(* CODESYS project util.library
   Company: TINEA
   Title: regulation
   Version: 0.0.0.0

Project tree, tasks and I/O mapping:
  libraries: Tc2_Standard, * (Beckhoff Automation GmbH)
  Data types/
    data type GEN_MODE
    data type POINT
  Global Variables/
    global variables Globale_Variablen
  POUs/
    analog monitors/
      function block HYSTERESIS [ST]
      function block LIMITALARM [ST]
    BCD CO_Nversions/
      function BCD_TO_INT [ST]
      function INT_TO_BCD [ST]
    bit_byte functions/
      function EXTRACT [ST]
      function PACK [ST]
      function PUTBIT [ST]
      function block UNPACK [ST]
    CO_Ntroller/
      function block PD [ST]
      function block PID [ST]
      function block PID_FIXCYCLE [ST]
    function manipulators/
      function block CHARCURVE [ST]
      function block RAMP_INT [ST]
      function block RAMP_REAL [ST]
    mathematical functions/
      function block DERIVATIVE [ST]
      function block INTEGRAL [ST]
      function block LIN_TRAFO [ST]
      function block STATISTICS_INT [ST]
      function block STATISTICS_REAL [ST]
      function block VARIANCE [ST]
    signals/
      function block BLINK [ST]
      function block FREQ_MEASURE [ST]
      function block GEN [ST]
    function Version_Util [ST]
  Visualizations/
*)

// Data types/GEN_MODE
TYPE GEN_MODE :
	(TRIANGLE:=0,TRIANGLE_POS:=1,SAWTOOTH_RISE:=2,SAWTOOTH_FALL:=3,RECTANGLE:=4,SINUS:=5,COSINUS:=6);
END_TYPE

// Data types/POINT
TYPE POINT :
STRUCT
	X,Y: DINT;
END_STRUCT
END_TYPE

// Global Variables/Globale_Variablen
{attribute 'Tc2GvlVarNames'}
VAR_GLOBAL
END_VAR

// POUs/BCD CO_Nversions/BCD_TO_INT
(* function reads BCD-Byte and returns its INT value; a wrong BCD value causes a return of -1 *)
FUNCTION BCD_TO_INT : INT
VAR_INPUT
	B:BYTE;		(* byte containing the BCD value *)
END_VAR

IF SHR(B,4)>9 OR B-SHL(SHR(B,4),4)>9 THEN
	BCD_TO_INT:=-1;
ELSE
	BCD_TO_INT:=B-SHR(B,4)*6;
END_IF;

END_FUNCTION

// POUs/signals/BLINK
FUNCTION_BLOCK BLINK
(* Function block to simulate a turn signal *)
VAR_INPUT
	ENABLE:BOOL;		(* TRUE:run Blink, FALSE: OUT keeps its value*)
	TIMELOW:TIME;		(* Time for OUT=FALSE *)
	TIMEHIGH:TIME;		(* Time for OUT=TRUE *)
END_VAR
VAR_OUTPUT
	OUT:BOOL;			(* output variable, starting with FALSE *)
END_VAR
VAR
	CLOCK:TP;
END_VAR

CLOCK();										(* call Timer *)
IF CLOCK.Q=FALSE AND ENABLE THEN	(* time passed or init *)
	CLOCK(IN:=FALSE);						(* reset Timer *)
	CLOCK(IN:=TRUE);						(* restart Timer *)
	IF OUT=FALSE THEN
		CLOCK.PT:=TIMEHIGH;
	ELSE
		CLOCK.PT:=TIMELOW;
	END_IF;
	OUT := NOT OUT;							(* invert *)
END_IF

END_FUNCTION_BLOCK

// POUs/function manipulators/CHARCURVE
(* function block to map an input signal on a characteristic curve *)
FUNCTION_BLOCK CHARCURVE
VAR_INPUT
	IN:INT;								(* input signal *)
	N:BYTE;							(* number of  points defining the characteristic curve : 2<=N<=11 *)
END_VAR
VAR_IN_OUT
	P:ARRAY[0..10] OF POINT;		(* ARRAY of N points to describe the characteristic curve *)
END_VAR
VAR_OUTPUT
	OUT:INT;							(* output variable *)
	ERR: BYTE;							(* error :
												0 : 	no error
												1 :	error in ARRAY: wrong sequence ( completely tested, only if IN is equal to largest X-value of P)
												2 :	IN outside of limits of P
												4 :	number of POINTS (N) invalid *)
END_VAR
VAR
	I:INT;
END_VAR

IF 1<N AND N<12 THEN							(* N zulässig ? *)
	ERR:=0;
	IF IN<P[0].X THEN							(* Prüfe, ob IN im zulässigen Bereich *)
		ERR:=2;
		OUT:=DINT_TO_INT(P[0].Y);
	ELSIF IN>P[N-1].X THEN						(* Prüfe, ob IN im zulässigen Bereich *)
		ERR:=2;
		OUT:=DINT_TO_INT(P[N-1].Y);
	ELSE
		FOR I:=1 TO N-1 DO
			IF P[I-1].X>=P[I].X THEN			(* Prüfe, ob Reihenfolge der Punkte richtig *)
				ERR:=1;
				EXIT;
			END_IF;
			IF IN<=P[I].X THEN					(* Verlasse Schleife, wenn IN im Intervall [I-1;I] *)
				EXIT;
			END_IF
		END_FOR;
		IF ERR=0 THEN
			OUT:=DINT_TO_INT(P[I].Y-(P[I].X-IN)*(P[I].Y-P[I-1].Y)/(P[I].X-P[I-1].X));	(* Berechne OUT *)
		ELSE
			OUT:=0;
		END_IF;
	END_IF
ELSE
	ERR:=4;
END_IF;

END_FUNCTION_BLOCK

// POUs/mathematical functions/DERIVATIVE
(* function block to approximate the derivative of a value *)
(* to calculate this, always four values are used in order to be as exact as possible *)
FUNCTION_BLOCK DERIVATIVE
VAR_INPUT
	IN:REAL;						(* input variable *)
	TM:DWORD;					(* time since last call in msec *)
	RESET:BOOL;					(* reset: set OUT to zero *)
END_VAR
VAR_OUTPUT
	OUT:REAL;					(* derivative *)
END_VAR
VAR
	X3,X2,X1:REAL;
	T2,T1:DWORD;
	INIT:BOOL:=TRUE;
END_VAR

IF INIT OR RESET THEN
	X1:=IN;
	X2:=IN;
	X3:=IN;
	OUT:=0;
	INIT:=FALSE;
ELSE
	IF TM>0 THEN
		OUT:=(3*(IN-X3)+X1-X2)/((3*T2+4*T1+3*TM))*1000;
		X3:=X2;
		X2:=X1;
		X1:=IN;
		T2:=T1;
		T1:=TM;
	END_IF;
END_IF;

END_FUNCTION_BLOCK

// POUs/bit_byte functions/EXTRACT
(* function returns Bit N of value X *)
FUNCTION EXTRACT : BOOL
VAR_INPUT
	X:DWORD;	(* value *)
	N:BYTE;		(* number of bit to be extracted *)
END_VAR
VAR
END_VAR

EXTRACT:=((SHR(X,N) AND 1)=1);

END_FUNCTION

// POUs/signals/FREQ_MEASURE
FUNCTION_BLOCK FREQ_MEASURE
(* FB to measure the frequency of a signal *)
VAR_INPUT
	IN:BOOL;						(* input signal *)
	PERIODS: INT (1..10) :=1;	(* out is the average frequency during PERIODS (number of periods) *)
	RESET: BOOL;				(* reset measurement *)
END_VAR
VAR_OUTPUT
	OUT:REAL;					(* frequency [Hz]*)
	VALID:BOOL;					(* FALSE: not yet PERIODS measurements done OR time distance between two rising edges > 3*OUT *)
END_VAR
VAR
	OLDIN: BOOL;
	INIT: BOOL;
	OLDT: TIME;
	DIFF: DWORD;
	ADIFF: ARRAY[0..9] OF DWORD;
	V: INT;
	B:INT;
	I: INT;
END_VAR

IF RESET THEN
	B:=0;
	V:=0;
	INIT:=FALSE;
	VALID:=FALSE;
	OUT:=0;
	RETURN;
END_IF

IF IN AND NOT OLDIN THEN	(*rising edge *)
	IF INIT THEN
		DIFF := TIME_TO_DWORD(TIME()-OLDT);
		IF Diff > 0 THEN
			ADIFF[B] := DIFF;
			B := (B+1) MOD PERIODS;
			V:= MIN(V+1, PERIODS);
			IF V=PERIODS THEN
				OUT := 0;
				FOR I:=0 TO PERIODS-1 DO
					OUT := OUT + ADIFF[I];
				END_FOR
				OUT := 1000.0 * PERIODS / OUT;
				VALID:=TRUE;
			ELSE
				VALID:=FALSE;
			END_IF
		END_IF
	END_IF
	INIT := TRUE;
	OLDT := TIME();
ELSIF INIT AND VALID AND TIME_TO_DWORD(TIME()-OLDT) > 3000*OUT THEN
	VALID:=FALSE;
	V:=0;
	B:=0;
END_IF

OLDIN:=IN;

END_FUNCTION_BLOCK

// POUs/signals/GEN
(* function block for generating some periodic functions *)
FUNCTION_BLOCK GEN
VAR_INPUT
	MODE:GEN_MODE;	(* define type :
								TRIANGLE				triangular	from - AMPL. to + AMPL.
								TRIANGLE_POS		triangular	from 0 to AMPL. 
								SAWTOOTH_RISE	sawtooth increasing from -AMPL. to +AMPL.
								SAWTOOTH_FALL	sawtooth decreasing from AMPL to -AMPL
								RECTANGLE			rectangular switching from  -AMPL. to +AMPL 
								SINUS					sinus
								COSINUS				cosinus *)
	BASE:BOOL;			(* FALSE: period referring to call; TRUE: period referring to time *)
	PERIOD:TIME:=t#1s;	(* period time, only relevant if BASE=TRUE *)
	CYCLES:INT:=1000;	(* number of calls per period, only relevant if BASE=FALSE *)
	AMPLITUDE:INT;		(* amplitude *)
	RESET:BOOL;			(* reset *)
END_VAR
VAR_OUTPUT
	OUT:INT;				(* generated function variable *)
END_VAR
VAR
	CET,PER:DINT;
	COUNTER:INT;
	CLOCK:TON;
	help: REAL;
END_VAR

IF RESET THEN
	COUNTER:=0;
	OUT:=0;
	CLOCK.PT := t#0s;
	CLOCK(IN:=FALSE);
ELSE
	IF BASE=FALSE THEN
		COUNTER:=(COUNTER+1)MOD CYCLES;
		CASE MODE OF
		0:	(* Dreiecksfunktion von -AMPL bis AMPL.*)
			OUT:=(CYCLES-2*ABS(CYCLES-2*COUNTER))*AMPLITUDE/CYCLES;
		1:	(* Dreiecksfunktion von 0 bis AMPL.*)
			OUT:=(CYCLES-ABS(CYCLES-2*COUNTER))*AMPLITUDE/CYCLES;
		2:	(* Sägezahn steigend *)
			OUT:=(2*COUNTER-CYCLES)*AMPLITUDE/CYCLES;
		3:	(* Sägezahn fallend *)
			OUT:=(CYCLES-2*COUNTER)*AMPLITUDE/CYCLES;
		4:	(* Rechteck AMPL./-AMPL. *)
			IF 2*COUNTER>CYCLES THEN
				OUT:=-AMPLITUDE;
			ELSE
				OUT:=AMPLITUDE;
			END_IF
		5:	(* Sinusfunktion *)
			help := 6.283167*COUNTER/CYCLES;
			OUT:=LREAL_TO_INT(SIN(help)*AMPLITUDE);
		6:	(* Cosinusfunktion *)
			help := 6.283167*COUNTER/CYCLES;
			OUT:=LREAL_TO_INT(COS(help)*AMPLITUDE);
		END_CASE;
	ELSE										(* Periodizität bzgl. Zeit *)
				CLOCK();									(* Timer abfragen *)
		IF CLOCK.PT<>PERIOD+PERIOD THEN			(* Initialisierung *)
			CLOCK.PT:=PERIOD+PERIOD;			(* Setze Timer auf zwei PERIODn *)
			CLOCK(IN:=TRUE);
		ELSE
			CET:=TIME_TO_DINT(CLOCK.ET);
			PER:=TIME_TO_DINT(PERIOD);
			IF CET>=PER THEN					(* Neuinitialisierung des Timers *)
				CLOCK(IN:=FALSE);
				CLOCK(IN:=TRUE);
				CET:=CET MOD PER;
			END_IF
			CASE MODE OF
			0:	(* Dreiecksfunktion -AMPL bis AMPL.*)
				OUT:=DINT_TO_INT((2*ABS(PER-2*CET)*AMPLITUDE+PER/2)/PER-AMPLITUDE);
			1:	(* Dreiecksfunktion 0 bis AMPL.*)
				OUT:=DINT_TO_INT(((PER-ABS(PER-2*CET))*AMPLITUDE+PER/2)/PER);
			2:	(* Sägezahn steigend *)
				OUT:=DINT_TO_INT((CET-PER)*2*AMPLITUDE/PER+AMPLITUDE);
			3:	(* Sägezahn fallend *)
				OUT:=DINT_TO_INT((PER-CET)*2*AMPLITUDE/PER+AMPLITUDE);
			4:	(* Rechteck AMPL./-AMPL. *)
				IF CET*2<PER THEN
					OUT:=-AMPLITUDE;
				ELSE
					OUT:=AMPLITUDE;
				END_IF
			5:	(* Sinusfunktion *)
				help := 6.283167*CET;
				help:=SIN(help/PER)*AMPLITUDE;
				OUT:=REAL_TO_INT(help+0.5);
			6:	(* Cosinusfunktion *)
				help := 6.283167*CET;
				help:=COS(help/PER)*AMPLITUDE;
				OUT:=LREAL_TO_INT(help+0.5);
			END_CASE;
		END_IF
	END_IF;
END_IF;

END_FUNCTION_BLOCK

// POUs/analog monitors/HYSTERESIS
(* function block, which sets OUT to TRUE, if input IN is less than LOW, and which sets OUT to FALSE, if input IN is bigger than HIGH *)
FUNCTION_BLOCK HYSTERESIS
VAR_INPUT
	IN:INT;			(* input value *)
	HIGH:INT;		(* upper threshold value *)
	LOW:INT;		(* lower threshold value *)
END_VAR
VAR_OUTPUT
	OUT:BOOL;	(* hysteresis value *)
END_VAR
VAR
END_VAR

IF  IN<LOW THEN
	OUT:=TRUE;
END_IF;
IF IN>HIGH THEN
	OUT:=FALSE;
END_IF;

END_FUNCTION_BLOCK

// POUs/BCD CO_Nversions/INT_TO_BCD
(* function reads INT and returns its BCD value; a wrong INT value (<0 or >99) causes a return of 255 *)
FUNCTION INT_TO_BCD : BYTE
VAR_INPUT
	I:INT;		(* INT value to be converted to BCD*)
END_VAR
VAR
END_VAR

IF I>99 OR I<0 THEN
	INT_TO_BCD:=255;
ELSE
	INT_TO_BCD:=INT_TO_BYTE((I/10)*6+I);
END_IF;

END_FUNCTION

// POUs/mathematical functions/INTEGRAL
(* function block to approximate the integral of IN over the time *)
FUNCTION_BLOCK INTEGRAL
VAR_INPUT
	IN:REAL;						(* input variable *)
	TM:DWORD;					(* time since last call in msec *)
	RESET:BOOL;					(* reset: OUT is set to zero and OVERFLOW to false *)
END_VAR
VAR_OUTPUT
	OUT:REAL;					(* value of the integral *)
	OVERFLOW:BOOL:=FALSE;	(* overflow *)
END_VAR
VAR
END_VAR

IF RESET THEN
	OUT:=0;
	OVERFLOW:=FALSE;
ELSIF NOT OVERFLOW  THEN
	IF 1E38 - IN*TM < OUT OR -1E38 - IN*TM > OUT THEN
		OVERFLOW:=TRUE;
	ELSE
		OUT:=OUT+IN*TM/1000;
	END_IF;
END_IF;

END_FUNCTION_BLOCK

// POUs/analog monitors/LIMITALARM
(* function block monitoring, whether the input value IN lies between LOW and HIGH *)
FUNCTION_BLOCK LIMITALARM
VAR_INPUT
	IN:INT;					(* INPUT value *)
	HIGH:INT;				(* upper threshold value *)
	LOW:INT;				(* lower threshold value *)
END_VAR
VAR_OUTPUT
	O:BOOL;				(* TRUE, if IN > HIGH, else FALSE *)
	U:BOOL;				(* TRUE, if IN < LOW, else FALSE *)
	IL:BOOL;				(* neither O nor U *)
END_VAR
VAR
END_VAR

O:=(IN>HIGH);
U:=(IN<LOW);
IL:=NOT (O OR U);

END_FUNCTION_BLOCK

// POUs/mathematical functions/LIN_TRAFO
(* linear transformation *)
FUNCTION_BLOCK LIN_TRAFO
VAR_INPUT
	IN: REAL;				(* input value*)
	IN_MIN:REAL;			(* minimum input value *)
	IN_MAX:REAL;			(* maximum input value *)
	OUT_MIN:REAL;		(* corresponding minimum output value *)
	OUT_MAX:REAL;		(* corresponding maximum output value *)
END_VAR
VAR_OUTPUT
	OUT: REAL;			(* output value *)
	ERROR: BOOL;		(* error: IN_MIN = IN_MAX or IN out of interval *)
END_VAR

VAR
	Diff: REAL;
END_VAR

Diff := IN_MAX-IN_MIN;
ERROR := (Diff=0) OR (IN<IN_MIN) OR (IN>IN_MAX);

IF NOT ERROR THEN
	OUT := (IN-IN_MIN)/Diff * (OUT_MAX-OUT_MIN) + OUT_MIN;
END_IF

END_FUNCTION_BLOCK

// POUs/bit_byte functions/PACK
(* pack eight bits into 1 byte *)
FUNCTION PACK : BYTE
VAR_INPUT
	B0:BOOL;		(* value of bit 0 *)
	B1:BOOL;		(* value of bit 1 *)
	B2:BOOL;		(* value of bit 2 *)
	B3:BOOL;		(* value of bit 3 *)
	B4:BOOL;		(* value of bit 4 *)
	B5:BOOL;		(* value of bit 5 *)
	B6:BOOL;		(* value of bit 6 *)
	B7:BOOL;		(* value of bit 7 *)
END_VAR

PACK:=BOOL_TO_BYTE(B7);
PACK:=PACK*2+BOOL_TO_BYTE(B6);
PACK:=PACK*2+BOOL_TO_BYTE(B5);
PACK:=PACK*2+BOOL_TO_BYTE(B4);
PACK:=PACK*2+BOOL_TO_BYTE(B3);
PACK:=PACK*2+BOOL_TO_BYTE(B2);
PACK:=PACK*2+BOOL_TO_BYTE(B1);
PACK:=PACK*2+BOOL_TO_BYTE(B0);

END_FUNCTION

// POUs/CO_Ntroller/PD
(* PD controller *)
FUNCTION_BLOCK PD
VAR_INPUT
	ACTUAL :REAL;		(* actual value, process variable *)
	SET_POINT:REAL;	(* desired value, set point *)
	KP:REAL;				(* proportionality const. (P)*)
	TV:REAL;				(* rate time, derivative time (D) in sec *)
	Y_MANUAL:REAL;		(* Y is set to this value as long as MANUAL=TRUE *)
	Y_OFFSET:REAL;		(* offset for manipulated variable *)
	Y_MIN:REAL;			(* minimum value for manipulated variable *)
	Y_MAX:REAL;			(* maximum value for manipulated variable *)
	MANUAL:BOOL;		(* 	TRUE: manual: Y is not influenced by controller,
								FALSE: controller determines Y *)
	RESET:BOOL;			(* reset: set Y output to Y_OFFSET *)
END_VAR
VAR_OUTPUT
	Y:REAL;				(* manipulated variable, set value*)
	LIMITS_ACTIVE:BOOL:=FALSE;	(* true set value would exceed limits Y_MIN, Y_MAX *)
END_VAR
VAR
	CLOCK:TON;
	D: DERIVATIVE;
	TMDIFF: DWORD;
	ERROR: REAL;
	INIT: BOOL:=TRUE;
	Y_ADDOFFSET: REAL;
	KPcopy:REAL;
	TVcopy:REAL;
END_VAR

IF KP<> 0 THEN
	ERROR := SET_POINT-ACTUAL;								(* Regeldifferenz *)

	IF RESET OR MANUAL OR INIT OR (KP<>KPcopy OR TV<>TVcopy) THEN							(* Reset oder Handbetrieb *)
		D(RESET:=TRUE);
		LIMITS_ACTIVE:=FALSE;
		IF RESET OR INIT THEN
			Y := Y_OFFSET;
			INIT:=FALSE;
			Y_ADDOFFSET :=  0;
		ELSIF MANUAL THEN
			Y := Y_MANUAL;
			Y_ADDOFFSET := Y_MANUAL-(Y_OFFSET+KP*(ERROR+D.OUT*TV));
		ELSE
			Y_ADDOFFSET := Y - Y_OFFSET - KP*ERROR;
		END_IF
		TMDIFF:=0;
		CLOCK(IN:=FALSE);									(* Timer neu starten *)
		CLOCK(PT:=t#1h, IN:=TRUE);

		TVcopy := TV;
		KPcopy := KP;
	ELSE
				CLOCK();												(* Timer abfragen *)
		TMDIFF:=TIME_TO_DWORD(CLOCK.ET);					(* Zeitdifferenz seit letztem Aufruf *)
	END_IF;

	IF TMDIFF>0 THEN
		CLOCK(IN:=FALSE);									(* Timer neu starten *)
		CLOCK(PT:=t#1h, IN:=TRUE);

		D(IN:=ERROR, TM:=TMDIFF, RESET:=FALSE);				(* Differential abschätzen *)

		Y:=Y_OFFSET+KP*(ERROR+D.OUT*TV) + Y_ADDOFFSET;

		LIMITS_ACTIVE:=FALSE;
		IF Y_MAX>Y_MIN AND Y>Y_MAX  THEN					(* Stellwert-Obergrenze überschritten *)
			Y:=Y_MAX;
			LIMITS_ACTIVE:=TRUE;
		END_IF;

		IF Y_MAX>Y_MIN AND Y<Y_MIN THEN						(* Stellwert-Untergrenze unterschritten *)
			Y:=Y_MIN;
			LIMITS_ACTIVE:=TRUE;
		END_IF;
	ELSE
		CLOCK(PT:=t#1h,IN:=TRUE);
	END_IF;

END_IF;

END_FUNCTION_BLOCK

// POUs/CO_Ntroller/PID
(* PD controller *)
FUNCTION_BLOCK PID
VAR_INPUT
	ACTUAL :REAL;		(* actual value, process variable *)
	SET_POINT:REAL;	(* desired value, set point *)
	KP:REAL;				(* proportionality const. (P)*)
	TN:REAL;				(* reset time (I) in sec *)
	TV:REAL;				(* rate time, derivative time (D) in sec*)
	Y_MANUAL:REAL;		(* Y is set to this value as long as MANUAL=TRUE *)
	Y_OFFSET:REAL;		(* offset for manipulated variable *)
	Y_MIN:REAL;			(* minimum value for manipulated variable *)
	Y_MAX:REAL;			(* maximum value for manipulated variable *)
	MANUAL:BOOL;		(* 	TRUE: manual: Y is not influenced by controller,
								FALSE: controller determines Y *)
	RESET:BOOL;			(* reset: set Y output to Y_OFFSET and reset integral part *)
END_VAR
VAR_OUTPUT
	Y:REAL;				(* manipulated variable, set value*)
	LIMITS_ACTIVE:BOOL:=FALSE;	(* true set value would exceed limits Y_MIN, Y_MAX *)
	OVERFLOW:BOOL:=FALSE;		(* overflow in integral part *)
END_VAR
VAR
	CLOCK:TON;
	I: INTEGRAL;
	D: DERIVATIVE;
	TMDIFF: DWORD;
	ERROR: REAL;
	INIT: BOOL:=TRUE;
	Y_ADDOFFSET: REAL;
	KPcopy:REAL;
	TNcopy:REAL;
	TVcopy:REAL;
END_VAR

IF TN>0 AND KP<> 0 AND (NOT OVERFLOW OR RESET OR MANUAL) THEN
	ERROR := SET_POINT-ACTUAL;								(* Regeldifferenz *)

	IF RESET OR MANUAL OR INIT OR (KP<>KPcopy OR TN<>TNcopy OR TV<>TVcopy) THEN							(* Reset oder Handbetrieb *)
		I(RESET:=TRUE);
		D(RESET:=TRUE);
		OVERFLOW:=FALSE;
		LIMITS_ACTIVE:=FALSE;
		IF RESET OR INIT THEN
			Y := Y_OFFSET;
			INIT:=FALSE;
			Y_ADDOFFSET := 0;
		ELSIF MANUAL THEN
			Y := Y_MANUAL;
			Y_ADDOFFSET := Y_MANUAL-(Y_OFFSET+KP*(ERROR+I.OUT/TN+D.OUT*TV));
		ELSE
			Y_ADDOFFSET := Y - Y_OFFSET - KP*ERROR;
		END_IF
		TMDIFF:=0;
		CLOCK(IN:=FALSE);									(* Timer neu starten *)
		CLOCK(PT:=t#1h, IN:=TRUE);

		TNcopy := TN;
		TVcopy := TV;
		KPcopy := KP;
	ELSE
				CLOCK();												(* Timer abfragen *)
		TMDIFF:=TIME_TO_DWORD(CLOCK.ET);					(* Zeitdifferenz seit letztem Aufruf *)
	END_IF;

	IF TMDIFF>0 THEN
		CLOCK(IN:=FALSE);									(* Timer neu starten *)
		CLOCK(PT:=t#1h, IN:=TRUE);

		D(IN:=ERROR, TM:=TMDIFF, RESET:=FALSE);				(* Differential abschätzen *)
		I(IN:=ERROR, TM:=TMDIFF, RESET:=FALSE);				(* Integral abschätzen *)

		OVERFLOW := I.OVERFLOW;
		IF NOT OVERFLOW THEN
			Y:=Y_OFFSET+KP*(ERROR+I.OUT/TN+D.OUT*TV) + Y_ADDOFFSET;
			IF Y>1E30 OR Y<-1E30 THEN						(* Overflow steht bevor, darf aber eigentlich nicht passieren *)
				OVERFLOW:=TRUE;
			END_IF;

			LIMITS_ACTIVE:=FALSE;
			IF Y_MAX>Y_MIN AND Y>Y_MAX  THEN				(* Stellwert-Obergrenze überschritten *)
				LIMITS_ACTIVE:=TRUE;
				IF KP<>0 THEN
					I(IN:=(Y_MAX-Y)*TN/KP,TM:=1000,RESET:=FALSE);		(* Integral korrigieren *)
				END_IF
				Y:=Y_MAX;
			END_IF;
			IF Y_MAX>Y_MIN AND Y<Y_MIN THEN					(* Stellwert-Untergrenze unterschritten *)
				LIMITS_ACTIVE:=TRUE;
				IF KP<>0 THEN
					I(IN:=(Y_MIN-Y)*TN/KP,TM:=1000,RESET:=FALSE);		(* Integral korrigieren *)
				END_IF
				Y:=Y_MIN;
			END_IF;
		END_IF;
	ELSE
		CLOCK(PT:=t#1h,IN:=TRUE);
	END_IF;

END_IF;

END_FUNCTION_BLOCK

// POUs/CO_Ntroller/PID_FIXCYCLE
(* PD controller *)
FUNCTION_BLOCK PID_FIXCYCLE
VAR_INPUT
	ACTUAL :REAL;		(* actual value, process variable *)
	SET_POINT:REAL;	(* desired value, set point *)
	KP:REAL;				(* proportionality const. (P)*)
	TN:REAL;				(* reset time (I) in sec *)
	TV:REAL;				(* rate time, derivative time (D) in sec*)
	Y_MANUAL:REAL;		(* Y is set to this value as long as MANUAL=TRUE *)
	Y_OFFSET:REAL;		(* offset for manipulated variable *)
	Y_MIN:REAL;			(* minimum value for manipulated variable *)
	Y_MAX:REAL;			(* maximum value for manipulated variable *)
	MANUAL:BOOL;		(* 	TRUE: manual: Y is not influenced by controller,
								FALSE: controller determines Y *)
	RESET:BOOL;			(* reset: set Y output to Y_OFFSET and reset integral part *)
	CYCLE:REAL;			(* time in s between two calls *)
END_VAR
VAR_OUTPUT
	Y:REAL;				(* manipulated variable, set value*)
	LIMITS_ACTIVE:BOOL:=FALSE;	(* true set value would exceed limits Y_MIN, Y_MAX *)
	OVERFLOW:BOOL:=FALSE;		(* overflow in integral part *)
END_VAR
VAR
	I: INTEGRAL;
	D: DERIVATIVE;
	TMDIFF: DWORD;
	ERROR: REAL;
	INIT: BOOL:=TRUE;
	Y_ADDOFFSET: REAL;
	KPcopy:REAL;
	TNcopy:REAL;
	TVcopy:REAL;
END_VAR

IF TN>0 AND KP<> 0 AND (NOT OVERFLOW OR RESET OR MANUAL) THEN
	ERROR := SET_POINT-ACTUAL;								(* Regeldifferenz *)

	IF RESET OR MANUAL OR INIT OR (KP<>KPcopy OR TN<>TNcopy OR TV<>TVcopy) THEN							(* Reset oder Handbetrieb *)
		I(RESET:=TRUE);
		D(RESET:=TRUE);
		OVERFLOW:=FALSE;
		LIMITS_ACTIVE:=FALSE;
		IF RESET OR INIT THEN
			Y := Y_OFFSET;
			INIT:=FALSE;
			Y_ADDOFFSET := 0;
		ELSIF MANUAL THEN
			Y := Y_MANUAL;
			Y_ADDOFFSET := Y_MANUAL-(Y_OFFSET+KP*(ERROR+I.OUT/TN+D.OUT*TV));
		ELSE
			Y_ADDOFFSET := Y - Y_OFFSET - KP*ERROR;
		END_IF
		TMDIFF:=0;

		TNcopy := TN;
		TVcopy := TV;
		KPcopy := KP;
	ELSE
		tmDiff:=REAL_TO_DWORD(CYCLE*1000);
	END_IF;

	IF TMDIFF>0 THEN

		D(IN:=ERROR, TM:=TMDIFF, RESET:=FALSE);				(* Differential abschätzen *)
		I(IN:=ERROR, TM:=TMDIFF, RESET:=FALSE);				(* Integral abschätzen *)

		OVERFLOW := I.OVERFLOW;
		IF NOT OVERFLOW THEN
			Y:=Y_OFFSET+KP*(ERROR+I.OUT/TN+D.OUT*TV) + Y_ADDOFFSET;
			IF Y>1E30 OR Y<-1E30 THEN						(* Overflow steht bevor, darf aber eigentlich nicht passieren *)
				OVERFLOW:=TRUE;
			END_IF;

			LIMITS_ACTIVE:=FALSE;
			IF Y_MAX>Y_MIN AND Y>Y_MAX  THEN				(* Stellwert-Obergrenze überschritten *)
				LIMITS_ACTIVE:=TRUE;
				IF KP<>0 THEN
					I(IN:=(Y_MAX-Y)*TN/KP,TM:=1000,RESET:=FALSE);		(* Integral korrigieren *)
				END_IF
				Y:=Y_MAX;
			END_IF;

			IF Y_MAX>Y_MIN AND Y<Y_MIN THEN					(* Stellwert-Untergrenze unterschritten *)
				LIMITS_ACTIVE:=TRUE;
				IF KP<>0 THEN
					I(IN:=(Y_MIN-Y)*TN/KP,TM:=1000,RESET:=FALSE);		(* Integral korrigieren *)
				END_IF
				Y:=Y_MIN;
			END_IF;
		END_IF;
	END_IF;

END_IF;

END_FUNCTION_BLOCK

// POUs/bit_byte functions/PUTBIT
(* function sets bit N of X to B and returns new value *)
FUNCTION PUTBIT : DWORD
VAR_INPUT
	X:DWORD;	(* value to be manipulated *)
	N:BYTE;		(* position of bit to be changed *)
	B:BOOL;		(* value of specified bit *)
END_VAR

IF B=TRUE THEN
	PUTBIT:=(X OR SHL(DWORD#1,N));
ELSE
	PUTBIT:=(X AND ROL(DWORD#4294967294,N));
END_IF;

END_FUNCTION

// POUs/function manipulators/RAMP_INT
(* function block to limit the slope of a value to a certain value *)
FUNCTION_BLOCK RAMP_INT
VAR_INPUT
	IN: INT;							(* input variable *)
	ASCEND: INT;						(* maximum positive slope *)
	DESCEND: INT;					(* maximum negative slope (non-negative!!) *)
	TIMEBASE: TIME;					(* reference for ASCEND/DESCEND :
											t#0s : ASCEND/DESCEND defined per call
											else : ASCEND/DESCEND defined per specified time*)
	RESET:BOOL;						(* reset *)
END_VAR
VAR_OUTPUT
	OUT: INT;							(* value of function with limited slope *)
END_VAR
VAR
	DIFF: DINT;
	OLD_IN: INT;
	TB,CET:DWORD;
	CH:INT;
	CLOCK: TON;
END_VAR

IF RESET=TRUE OR CLOCK.PT<>TIMEBASE THEN			(* Reset *)
	OLD_IN:=IN;
	CLOCK(PT:=TIMEBASE,IN:=FALSE);
END_IF

DIFF:=INT_TO_DINT(IN)-OLD_IN;									(* Änderung zum letzten WERT *)

IF TIMEBASE=t#0s THEN								(* Bezugswert : Aufruf *)
	IF DIFF>ASCEND THEN
		OUT:=OLD_IN+ASCEND;
	ELSIF DIFF<-DESCEND THEN
		OUT:=OLD_IN-DESCEND;
	ELSE
		OUT:=IN;
	END_IF;
ELSE												(* Bezugswert : TIMEBASE *)
	TB:=TIME_TO_DWORD(TIMEBASE);					(* TIMEBASE als DWORD *)
		CLOCK();
	CET:=TIME_TO_DWORD(CLOCK.ET);					(* verstrichene Zeit *)
	IF CET>0 THEN									(* wenn Zeit verstrichen *)
		IF (DWORD_TO_DINT(TB)*DIFF+CET/2)/DWORD_TO_DINT(CET)>ASCEND THEN			(* zu starker Anstieg *)
			CH:=DWORD_TO_INT((CET*ASCEND)/TB);
			IF CH<>0 THEN
					OUT:=OLD_IN+CH;
			END_IF;
		ELSIF DIFF*TB/DWORD_TO_DINT(CET)<-DESCEND THEN	(* zu starker Abfall *)
			CH:=DWORD_TO_INT((CET*DESCEND)/TB);
			IF CH<>0 THEN
					OUT:=OLD_IN-CH;
			END_IF;
		ELSE
			CH:=1;									(* Änderung in erlaubten Grenzen *)
			OUT:=IN;
		END_IF;
		IF CH<>0 THEN
			CLOCK(IN:=FALSE);						(* Timer neu starten *)
			CLOCK(IN:=TRUE);
		END_IF;
	ELSE											(* keine Zeit verstrichen *)
		CLOCK.PT:=TIMEBASE;							(* => ggf. Initialisierung *)
		CLOCK(IN:=TRUE);							(* => ggf. Timer neu starten *)
	END_IF;
END_IF;

OLD_IN:=OUT;

END_FUNCTION_BLOCK

// POUs/function manipulators/RAMP_REAL
(* function block to limit the slope of a value to a certain value *)
FUNCTION_BLOCK RAMP_REAL
VAR_INPUT
	IN: REAL;							(* input variable *)
	ASCEND: REAL;					(* maximum positive slope *)
	DESCEND: REAL;				(* maximum negative slope (non-negative!!) *)
	TIMEBASE: TIME;					(* reference for ASCEND/DESCEND :
											t#0s : ASCEND/DESCEND defined per call
											else : ASCEND/DESCEND defined per specified time*)
	RESET:BOOL;						(* reset *)
END_VAR
VAR_OUTPUT
	OUT: REAL;						(* value of function with limited slope *)
END_VAR
VAR
	DIFF: REAL;
	OLD_IN: REAL;
	TB,CET:DWORD;
	CLOCK: TON;
	probe:REAL;
END_VAR

IF RESET=TRUE OR CLOCK.PT<>TIMEBASE THEN			(* Reset *)
	OLD_IN:=IN;
	CLOCK(PT:=TIMEBASE,IN:=FALSE);
END_IF

DIFF:=IN-OLD_IN;									(* Änderung zum letzten WERT *)

IF TIMEBASE=t#0s THEN								(* Bezugswert : Aufruf *)
	IF DIFF>ASCEND THEN
		OUT:=OLD_IN+ASCEND;
	ELSIF DIFF<-DESCEND THEN
		OUT:=OLD_IN-DESCEND;
	ELSE
		OUT:=IN;
	END_IF;
ELSE												(* Bezugswert : TIMEBASE *)
	TB:=TIME_TO_DWORD(TIMEBASE);					(* TIMEBASE als DWORD *)
		CLOCK();
	CET:=TIME_TO_DWORD(CLOCK.ET);					(* verstrichene Zeit *)
	IF CET>0 THEN									(* wenn Zeit verstrichen *)
		CLOCK(IN:=FALSE);							(* Timer neu starten *)
		CLOCK(IN:=TRUE);
		probe:=DIFF*TB/CET;
		IF probe>ASCEND THEN						(* zu starker Anstieg *)
			OUT:=OLD_IN+ASCEND*CET/DWORD_TO_REAL(TB);
		ELSIF probe<-DESCEND THEN					(* zu starker Abfall *)
			OUT:=OLD_IN-DESCEND*CET/DWORD_TO_REAL(TB);
		ELSE										(* Änderung in erlaubten Grenzen *)
			OUT:=IN;
		END_IF;
	ELSE											(* keine Zeit verstrichen *)
		CLOCK.PT:=TIMEBASE;							(* => ggf. Initialisierung *)
		CLOCK(IN:=TRUE);							(* => ggf. Timer neu starten *)
	END_IF;
END_IF;

OLD_IN:=OUT;

END_FUNCTION_BLOCK

// POUs/mathematical functions/STATISTICS_INT
(* function block for statistics: calculating minimum, maximum and average of an input value *)
FUNCTION_BLOCK STATISTICS_INT
VAR_INPUT
	IN: INT;				(* input value*)
	RESET: BOOL;		(* reset: average set to 0, min and max to minimum and maximum possible INTs*)
END_VAR
VAR_OUTPUT
	MN: INT:=32767;		(* minimum value*)
	MX: INT:=-32768;		(* maximum value*)
	AVG: INT;				(* average value*)
END_VAR
VAR
	SUM:DINT;
	COUNTER:DINT;
END_VAR

IF RESET THEN
	AVG:=IN;
	COUNTER:=0;
	SUM:=0;
	MN:=IN;
	MX:=IN;
ELSE
	IF IN<MN THEN
		MN:=IN;
	END_IF
	IF IN>MX THEN
		MX:=IN;
	END_IF
	IF ABS(SUM)>2000000000 OR ABS(COUNTER)>2000000000 THEN		(* falls Überlauf droht *)
		SUM:=SUM/2;
		COUNTER:=COUNTER/2;
	END_IF;

	COUNTER:=COUNTER+1;
	SUM:=SUM+IN;
	AVG:=DINT_TO_INT((SUM+COUNTER/2)/COUNTER);  				(* gerundeter Durchschnitt *)
END_IF;

END_FUNCTION_BLOCK

// POUs/mathematical functions/STATISTICS_REAL
(* function block for statistics: calculating minimum, maximum and average of an input value *)
FUNCTION_BLOCK STATISTICS_REAL
VAR_INPUT
	IN: REAL;					(* input value*)
	RESET: BOOL;			(* reset: average set to 0, min and max to minimum and maximum possible REALs*)
END_VAR
VAR_OUTPUT
	MN: REAL:=3E+38;		(* minimum value*)
	MX: REAL:=1E-37;			(* maximum value*)
	AVG: REAL;				(* average value*)
END_VAR
VAR
	COUNTER: DINT;
	SUM:REAL;
END_VAR

IF RESET THEN
	AVG:=0;
	COUNTER:=0;
	SUM:=0;
	MN:=3.402823466e+38;
	MX:=1.175494351e-38;
ELSE
	IF IN<MN THEN
		MN:=IN;
	END_IF
	IF IN>MX THEN
		MX:=IN;
	END_IF

	IF ABS(COUNTER)>2000000000 THEN						(* falls Überlauf droht *)
		COUNTER:=COUNTER/2;
	END_IF;

	COUNTER:=COUNTER+1;
	AVG:=AVG/COUNTER*(COUNTER-1)+IN/COUNTER;
END_IF;

END_FUNCTION_BLOCK

// POUs/bit_byte functions/UNPACK
(* function block unpacks byte into 8 bits *)
FUNCTION_BLOCK UNPACK
VAR_INPUT
	B:BYTE;	(* byte to be unpacked *)
END_VAR
VAR_OUTPUT
	B0:BOOL;		(* value of bit 0 *)
	B1:BOOL;		(* value of bit 1 *)
	B2:BOOL;		(* value of bit 2 *)
	B3:BOOL;		(* value of bit 3 *)
	B4:BOOL;		(* value of bit 4 *)
	B5:BOOL;		(* value of bit 5 *)
	B6:BOOL;		(* value of bit 6 *)
	B7:BOOL;		(* value of bit 7 *)
END_VAR
VAR
END_VAR

B7:=BYTE_TO_BOOL(B AND 128);
B6:=BYTE_TO_BOOL(B AND 64);
B5:=BYTE_TO_BOOL(B AND 32);
B4:=BYTE_TO_BOOL(B AND 16);
B3:=BYTE_TO_BOOL(B AND 8);
B2:=BYTE_TO_BOOL(B AND 4);
B1:=BYTE_TO_BOOL(B AND 2);
B0:=BYTE_TO_BOOL(B AND 1);

END_FUNCTION_BLOCK

// POUs/mathematical functions/VARIANCE
(* function block to calculate the mathematical variance of a variable*)
FUNCTION_BLOCK VARIANCE
VAR_INPUT
	IN:REAL;		(* input variable *)
	RESET:BOOL;	(* reset *)
END_VAR
VAR_OUTPUT
	OUT:REAL;	(* variance *)
END_VAR
VAR
	Z:INT;
	A,B:REAL;
END_VAR

IF RESET THEN
	Z:=0;
	A:=0;
	B:=0;
	OUT:=0;
ELSE
	Z:=Z+1;
	A:=A+IN*IN;
	B:=B+IN;
	OUT:=(A-B*B/Z)/Z;
END_IF;

END_FUNCTION_BLOCK

// POUs/Version_Util
FUNCTION Version_Util : WORD
VAR_INPUT
	B:BOOL;
END_VAR
VAR
END_VAR
(******************************************************************************************)
(* Version,  Datum	Kommentar											*)
(* 1.00	28.02.2001	generated								 			*)
(* 1.01	29.06.2001	bugfix in GEN (HP)									*)
(* 1.02	03.01.2002	INTEGRAL was calculated for sec instead of msec 	*)
(* 1.03 	12.11.2002	comments added *)
(* 1.04 	23.01.2003	GEN:initial values for PERIOD and CYCLES to avoid div by zero *)
(* 1.05	13.06.2003	DERIVATIVE was calculated for sec instead of msec *)
(*	ATTENTION		TV/TN inputs of PD and PID refer to sec instead of msec *)
(* 1.06	25.06.2003	PD/PID: input Y_MANUAL added *)
(* 1.07	13.10.2003	PID_FIXCYCLE added *)
(* 1.08	09.01.2004	CHARCURVE: overflow fixed *)
(* 1.09	30.01.2004	GEN: if time based, reset induced freeze *)
(* 1.10	12.02.2004	all libs except standard.lib removed *)
(* 1.11	11.03.2005	PID: avoid jumps in Y (when limits change) by correcting integral part ; LIN_TRAFO added*)
(* 1.12	14.03.2005	FREQ_MEASURE added *)
(* 1.13	16.06.2005	PID/PID_FIXCYCLE/PD: no jumps when KP/TN/TV are changing (#4777) *)
(* 1.14	23.08.2006	#5709: Datatype overflow in RAMP_INT *)
(* 1.15	16.05.2007	Typed literal warnings removed (bug #7576)*)
(* 1.16	18.05.2010	Too complex expression for SH removed (bug #9780)*)
(******************************************************************************************)

Version_Util := 116;

END_FUNCTION
